PROGRAM MAIN
VAR
	fbTransport: TransportSystem('MAIN.TPS_A');
END_VAR

END_PROGRAM

(* stored: Version 1.1.0.1, ProductVersion 3.1.4024.3
   POU MAIN: Id {b807fc2e-1114-4564-88f5-927cd81451cd}, SpecialFunc None *)
